FUNCTION_BLOCK FB_HMIEButton EXTENDS FB_BaseComponent IMPLEMENTS ITF_HMIEButton
VAR
	bContact			: BOOL;
	bActive				: BOOL;	//wybrany
	bVisible			: BOOL; //widoczny
	bEnable				: BOOL; //wlaczony
END_VAR

METHOD PUBLIC IsActive : BOOL
VAR_INPUT
END_VAR
IsActive		:= THIS^.bActive;
END_METHOD

METHOD PUBLIC IsEnable : BOOL
VAR_INPUT
END_VAR
IsEnable		:= THIS^.bEnable;
END_METHOD

METHOD PUBLIC IsPressed : BOOL
VAR_INPUT
END_VAR
IsPressed		:= THIS^.bContact;
END_METHOD

METHOD PUBLIC IsVisible : BOOL
VAR_INPUT
END_VAR
IsVisible		:= THIS^.bVisible;
END_METHOD

METHOD PUBLIC SetActive
VAR_INPUT
	bIN: BOOL;
END_VAR
THIS^.bActive		:= bIN;
END_METHOD

METHOD PUBLIC SetEnable
VAR_INPUT
	bIN: BOOL;
END_VAR
THIS^.bEnable		:= bIN;
END_METHOD

METHOD PUBLIC SetPressed
VAR_INPUT
	bIN: BOOL;
END_VAR
THIS^.bContact		:= bIN;
END_METHOD

METHOD PUBLIC SetVisible
VAR_INPUT
	bIN: BOOL;
END_VAR
THIS^.bVisible		:= bIN;
END_METHOD

END_FUNCTION_BLOCK

(* stored: Version 1.1.0.1
   POU FB_HMIEButton: Id {936d0e57-6045-41ed-8f87-65656e00bc73}, SpecialFunc None
   Method IsActive: Id {582562ff-b9de-4d7d-a44e-ecab9d1d0a4b}
   Method IsEnable: Id {cc02517e-7fb6-47a3-8cdf-80218cb01ab6}
   Method IsPressed: Id {4bba51f0-58a8-4445-82db-fb1d08a086cc}
   Method IsVisible: Id {a6226b79-41e0-467b-aa0a-501eef35b9b4}
   Method SetActive: Id {bc4aabf8-0a33-46b0-83fb-083bcdcc6795}
   Method SetEnable: Id {b4464f1e-1039-4330-a435-f23826a59a2f}
   Method SetPressed: Id {f64a26bb-2bd6-4352-9080-c9b29385f5a8}
   Method SetVisible: Id {ae3fd991-7f0d-4cc8-be08-e9c95a3ba73e} *)
